(* CODESYS project wago_mysql_example_v0.0.1.ecp

Project tree, tasks and I/O mapping:
  PFC200_CS_2ETH_RS : 750-8202 PFC200 2ETH RS, WAGO, order no. 0750-8202, version 5.11.1.16
    application Application
      libraries: ; WagoAppSQL_MySQL, * (WAGO); WagoSysErrorBase, * (WAGO); VisuDialogs, * (System); WagoSysString, * (WAGO)
      task PLC_Task (cyclic, interval t#10ms, priority 14) calls PLC_PRG
      task VISU_TASK (cyclic, interval 100 ms, priority 15) calls VisuElems.Visu_Prg
      program PLC_PRG [ST]
      function funMySqlinsertStatement [ST]
      visualisation Visualization
      function funSqlResultToString [ST]
    DeviceAdapter
    Kbus : Kbus, WAGO, version 1.4.0.2
        unmapped channels: K-BUS diagnostics
      _16_DI_Generic : 075x-16DI, WAGO, order no. 075x-16DI, version 0.0.0.13
          settings: K-BUS Module slot index = 1
          unmapped channels: _IN
        DeviceAdapter
      _16_DO_Generic : 075x-16DO, WAGO, order no. 075x-16DO, version 0.0.0.13
          settings: K-BUS Module slot index = 2
          unmapped channels: _OUT
        DeviceAdapter
    MODBUS
      MODBUS : MODBUS, WAGO, order no. n/a, version 1.1.1.15
    Serial
      COM1 : COM1, WAGO, version 0.0.0.19
  libraries: VisuSymbols, 3.5.10.0 (System); WagoVisuIcons, 1.0.0.8 (WAGO)
  text list GlobalTextList
*)

// PFC200_CS_2ETH_RS/Application/PLC_PRG
PROGRAM PLC_PRG
VAR
	(* example project to query and insert data into SQL table *)
	(* written by : Jesse Cox @ WAGO USA jesse.cox@wago.com *)
	/// function blocks
	fbMySqlLogin		: FbMySql_Login;
	fbMySqlExecute		: FbMySql_Execute;
	fbMySqlQuery		: FbMySql_Query;
	fbMySqlLogout		: FbMySql_Logout;
	
	// login variables
	sMySqlHost			: STRING := '<yourServerIP>';
	uiMySqlPort			: UINT := 3306;
	sMySqlUsername		: STRING := '<username>';
	sMySqlPassword		: STRING := '<password>';
	sMySqlDB			: STRING := 'databaseName';
	xMySqlLogin			: BOOL;
	xMySqlLoginBusy		: BOOL;
	xMySqlLoginError	: BOOL;
	oMySqlLoginStatus	: WagoSysErrorBase.FbResult;
	sMySqlLoginStatus	: STRING(200);
	xMySqlIsConnected	: BOOL;
	
	// execute INSERT variables
	aMySqlInsetStatement: ARRAY [0..MYSQL_SQL_UPPER_BOUND] OF STRING(MYSQL_SQL_LENGTH);
	xMySqlExecute		: BOOL;
	xMySqlExecuteBusy	: BOOL;
	xMySqlExecuteError	: BOOL;
	oMySqlExecuteStatus	: WagoSysErrorBase.FbResult;
	sMySqlExecuteStatus	: STRING(200);
	
	// execute QUERY variables
	aMySqlQueryStatement: ARRAY [0..MYSQL_SQL_UPPER_BOUND] OF STRING(MYSQL_SQL_LENGTH);
	xMySqlQuery			: BOOL;
	typMySqlQueryRslt	: typMySql_ResultSet;
	xMySqlQueryBusy		: BOOL;
	xMySqlQueryError	: BOOL;
	oMySqlQueryStatus	: WagoSysErrorBase.FbResult;
	sMySqlQueryStatus	: STRING(200);
	
	// logout	
	xMySqlLogout		: BOOL;
	xMySqlLogoutBusy	: BOOL;
	xMySqlLogoutError	: BOOL;
	oMySqlLogoutStatus	: WagoSysErrorBase.FbResult;
	sMySqlLogoutStatus	: STRING(200);
	
	
	// my values
	sMySqlTable			: STRING := 'WagoTestTable';
	myVal1				: WORD := 99;
	myVal2				: WORD := 375;
	myResults			: ARRAY[0..100] OF STRING;
END_VAR

fbMySqlLogin(
	sHost:= sMySqlHost, 
	uiPort:= uiMySqlPort, 
	sUsername:= sMySqlUsername, 
	sPassword:= sMySqlPassword, 
	sDatabase:= sMySqlDB, 
	xTrigger:= xMySqlLogin, 
	xBusy=> xMySqlLoginBusy, 
	xError=> xMySqlLoginError, 
	oStatus=> oMySqlLoginStatus, 
	sStatus=> sMySqlLoginStatus, 
	xConnected=> xMySqlIsConnected);

	// create the INSERT statement from function
aMySqlInsetStatement := funMySqlinsertStatement(sTable:= sMySqlTable, Val1:= myVal1, Val2:= myVal2);

fbMySqlExecute(
	aSqlCommand:= aMySqlInsetStatement, 
	xTrigger:= xMySqlExecute, 
	xBusy=> xMySqlExecuteBusy, 
	xError=> xMySqlExecuteError, 
	oStatus=> oMySqlExecuteStatus, 
	sStatus=> sMySqlExecuteStatus);

	// create the QUERY statement 	
aMySqlQueryStatement[0] := 'SELECT * FROM WagoTestTable';

fbMySqlQuery(
	aSqlCommand:= aMySqlQueryStatement, 
	xTrigger:= xMySqlQuery, 
	typResultSet:= typMySqlQueryRslt, 
	xBusy=> xMySqlQueryBusy, 
	xError=> xMySqlQueryError, 
	oStatus=> oMySqlQueryStatus, 
	sStatus=> sMySqlQueryStatus);
	
myResults := funSqlResultToString(tySQLResults:= typMySqlQueryRslt);
	
fbMySqlLogout(
	xTrigger:= xMySqlLogout, 
	xBusy=> xMySqlLogoutBusy, 
	xError=> xMySqlLogoutError, 
	oStatus=> oMySqlLogoutStatus, 
	sStatus=> sMySqlLogoutStatus);

END_PROGRAM

// PFC200_CS_2ETH_RS/Application/funMySqlinsertStatement
FUNCTION funMySqlinsertStatement : ARRAY [0..MYSQL_SQL_UPPER_BOUND] OF STRING(MYSQL_SQL_LENGTH);
VAR_INPUT
	sTable		: STRING;
	Val1		: WORD;
	Val2		: WORD;
END_VAR
VAR
	sInsertStatementHold		: ARRAY [0..MYSQL_SQL_UPPER_BOUND] OF STRING(MYSQL_SQL_LENGTH);
END_VAR

//*********************************************************************
// example: INSERT INTO myTableName (Val1, Val2) VALUES (myVal1, myVal2)
//*********************************************************************

sInsertStatementHold[0] := 'INSERT INTO ';
sInsertStatementHold[1] := sTable;
sInsertStatementHold[2] := '(Val1, Val2) VALUES (';
sInsertStatementHold[3] := WORD_TO_STRING(Val1);
sInsertStatementHold[4] := ', ';
sInsertStatementHold[5] := WORD_TO_STRING(Val2);
sInsertStatementHold[6] := ')';

funMySqlinsertStatement := sInsertStatementHold;

END_FUNCTION

// PFC200_CS_2ETH_RS/Application/funSqlResultToString
FUNCTION funSqlResultToString : ARRAY[0..100] OF STRING
VAR_INPUT
	tySQLResults	: typMySql_ResultSet;
END_VAR
VAR
	i				: INT;
	x				: INT;
END_VAR

FOR i := 0 TO tySQLResults.uiRowCount DO
	FOR x := 0 TO 100 DO
		funSqlResultToString[i] := CONCAT(funSqlResultToString[i], ASCIIBYTE_TO_STRING(tySQLResults.abRows[i][x]));
	END_FOR
END_FOR

END_FUNCTION

// PFC200_CS_2ETH_RS/Application/Visualization
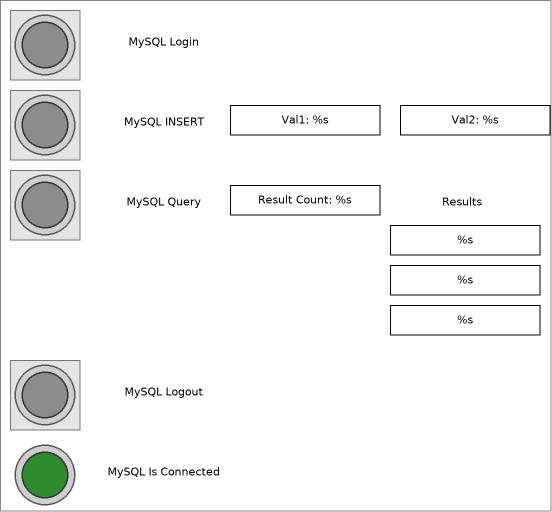
VISUALIZATION Visualization  // 552x512
    PushSwitch (10,10 70x70), variable: PLC_PRG.xMySqlLogin, behaviour: TOGGLE, style: Switch-PushSwitch-Gray
    PushSwitch (10,90 70x70), variable: PLC_PRG.xMySqlExecute, behaviour: TOGGLE, style: Switch-PushSwitch-Gray
    PushSwitch (10,170 70x70), variable: PLC_PRG.xMySqlQuery, behaviour: TOGGLE, style: Switch-PushSwitch-Gray
    PushSwitch (10,360 70x70), variable: PLC_PRG.xMySqlLogout, behaviour: TOGGLE, style: Switch-PushSwitch-Gray
    Lamp1 (10,440 70x70), variable: PLC_PRG.xMySqlIsConnected, style: Lamp-Lamp1-Green
    Label (89,27 150x30), "MySQL Login"
    Label (89,107 150x30), "MySQL INSERT"
    Label (89,187 150x30), "MySQL Query"
    Label (89,377 150x30), "MySQL Logout"
    Label (89,457 150x30), "MySQL Is Connected"
    Rectangle (230,105 150x30), "Val1: %s", text variable: PLC_PRG.myVal1
        OnMouseDown: write the text variable via VisuDialogs.Numpad
    Rectangle (400,105 150x30), "Val2: %s", text variable: PLC_PRG.myVal2
        OnMouseClick: write the text variable via VisuDialogs.Numpad
    Rectangle (230,185 150x30), "Result Count: %s", text variable: PLC_PRG.typMySqlQueryRslt.uiRowCount
    Rectangle (390,225 150x30), "%s", text variable: PLC_PRG.myResults[0]
    Rectangle (390,265 150x30), "%s", text variable: PLC_PRG.myResults[1]
    Rectangle (390,305 150x30), "%s", text variable: PLC_PRG.myResults[2]
    Label (389,187 150x30), "Results"
END_VISUALIZATION
